FUNCTION_BLOCK FINAL FB_StepEngine EXTENDS FB_EventLogger  
VAR_INPUT
	Size					: UINT;
	Flags					: DWORD;
END_VAR             		
VAR_IN_OUT 
	Control					: ST_System;
	StepDesc				: ARRAY[*] OF STRING;
	MatrixA					: ARRAY[*] OF DINT;
	MatrixB					: ARRAY[*] OF DINT;
	MatrixC					: ARRAY[*] OF DINT;
	MatrixD					: ARRAY[*] OF DINT;
	TimerSP					: ARRAY[*] OF REAL;         		
END_VAR  
VAR_OUTPUT          		
	Outputs					: ARRAY[0..3] OF DINT; 
END_VAR             		
VAR      
	_StepReq				: INT;
	_DeviceAlarm			: BOOL;      		
	_SeqInterface			: ST_SequenceInterface;         		
	_StepTimeDn				: BOOL;
	_StepTimeRun			: BOOL;
	_StepChanged			: BOOL;
	_Disabled				: BOOL;
	_StepNum				: INT;
	_StepNumChan			: INT;
	_StepNumPrev			: INT;
	_StepTime_ET			: REAL;
	_StepTime_ETDT			: TIME;
	_StepTimeLeft			: REAL;
	_StepTimeLeftDT			: TIME;
	_StepTimePrev_ET		: REAL;
	_Message				: STRING;
	_Alarm					: BOOL;	
	_AlarmNum				: DINT;					
	_Fault					: BOOL;									
	_CurrentStep			: ARRAY[0..255] OF BOOL;
	_HistoryIndex			: INT;
END_VAR             		
VAR PERSISTENT      	
	_Name					: STRING[15];				
	_Description			: STRING[40];	
	_Disable				: BOOL;   			
	_AlarmMute				: BOOL;						
	_StepTime_PT			: REAL;
	_LastActiveStep			: INT;
	_History				: ARRAY[0..99] OF ST_SequenceHistory;	
	_Variables				: ARRAY [0..9] OF ST_Variable;									
END_VAR

M_AlarmMonitor();
F_CheckIndexBounds(0,UINT_TO_INT(Size),_StepNum);
F_CheckIndexBounds_REAL(0,65534,_StepTime_ET);
F_CheckIndexBounds_REAL(0,65534,_StepTime_PT);
F_CheckIndexBounds_REAL(0,65534,_StepTimeLeft);

IF  _Disable THEN
	_StepNum := 0;
	_Disabled := TRUE;
	_Message := 'Sequence Disabled';
ELSE
	_StepNum := _StepReq;
	_Disabled := FALSE;
	_Message:= StepDesc[_StepNum];
END_IF

IF Control.PackMLState.Complete THEN
	_LastActiveStep := 0;
END_IF

Outputs[0] := MatrixA[_StepNum];
Outputs[1] := MatrixB[_StepNum];
Outputs[2] := MatrixC[_StepNum];
Outputs[3] := MatrixD[_StepNum];

MEMSET(destAddr:= ADR(_CurrentStep), fillByte:= 0, n:= SIZEOF(_CurrentStep));
_CurrentStep[_StepNum] := TRUE;

IF _StepChanged THEN
	_StepTime_PT := TimerSP[_StepNum];
END_IF

_StepTime_ET := _StepTime_ET + Control.SystemTime.ScanTime;
_StepTime_ETDT := REAL_TO_TIME(_StepTime_ET);

IF _StepNum <> _StepNumChan THEN
	_StepTimePrev_ET := _StepTime_ET;
	_StepTime_ET := 0;
	_StepNumPrev := _StepNumChan;
	IF MatrixA[_StepNumChan].31 = TRUE THEN _LastActiveStep := _StepNumChan; END_IF
	IF MatrixA[_StepNumChan].30 = TRUE THEN _LastActiveStep := 0; END_IF	
	_StepNumChan := _StepNum;
	_StepChanged := TRUE;
	_StepTimeDn := FALSE;	
ELSE
	IF _StepTime_ET <= _StepTime_PT THEN
		_StepTimeLeft := _StepTime_PT - _StepTime_ET;
		_StepTimeLeftDT := REAL_TO_TIME(_StepTimeLeft);
	ELSE
		_StepTimeDn := TRUE;
	END_IF
	_StepChanged := FALSE;	
END_IF

IF _StepTime_PT = 0 THEN
	_StepTimeLeft := 0;
	_StepTimeLeftDT := REAL_TO_TIME(_StepTimeLeft);
END_IF

_History[0].StepNum:= _StepNum;
_History[0].StepTime:= _StepTime_ET;
_History[0].Message:= _Message;
	
IF _StepNumPrev <> _History[1].StepNum THEN 
	FOR _historyIndex:= 99 TO 2 BY -1 DO
		_History[F_CheckIndexBounds(0,99,_historyIndex)]:= _History[F_CheckIndexBounds(0,99,_historyIndex)-1];
	END_FOR
	_History[1].StepNum:= _StepNumPrev;
	_History[1].StepTime:= _StepTimePrev_ET;
	_History[1].Message:= StepDesc[_StepNumPrev];
END_IF

{attribute 'monitoring' := 'variable'}
PROPERTY PUBLIC Alarm : Bool
GET
Alarm := _Alarm;
END_GET
END_PROPERTY

{attribute 'monitoring' := 'variable'}
PROPERTY PUBLIC AlarmMute : BOOL
SET
AlarmMute := _AlarmMute;
END_SET
END_PROPERTY

{attribute 'monitoring' := 'variable'}
PROPERTY PUBLIC CurrentStep : REFERENCE TO ARRAY[0..255] OF BOOL
GET
CurrentStep REF= _CurrentStep;
END_GET
END_PROPERTY

{attribute 'monitoring' := 'variable'}
PROPERTY PUBLIC Description : String[40]
GET
Description := _Description;
END_GET
SET
_Description := Description;
END_SET
END_PROPERTY

{attribute 'monitoring' := 'variable'}
PROPERTY PUBLIC DeviceAlarm : BOOL
GET
DeviceAlarm :=_DeviceAlarm;
END_GET
SET
_DeviceAlarm := DeviceAlarm;
END_SET
END_PROPERTY

{attribute 'monitoring' := 'variable'}
PROPERTY PUBLIC Disable : BOOL
SET
_Disable := Disable;
END_SET
END_PROPERTY

{attribute 'monitoring' := 'variable'}
PROPERTY PUBLIC Disabled : BOOL
GET // PUBLIC
Disabled := _Disabled;
END_GET
SET
_Disabled := Disabled;
END_SET
END_PROPERTY

{attribute 'monitoring' := 'variable'}
PROPERTY PUBLIC Fault : Bool
SET
_Fault := Fault;
END_SET
END_PROPERTY

PROPERTY PUBLIC History :REFERENCE to ARRAY[0..99] OF ST_SequenceHistory
GET
History REF=_History;
END_GET
END_PROPERTY

{attribute 'monitoring' := 'variable'}
PROPERTY PUBLIC LastActiveStep : int
GET // PUBLIC
LastActiveStep := _LastActiveStep;
END_GET
SET
_LastActiveStep := LastActiveStep;
END_SET
END_PROPERTY

METHOD PROTECTED M_AlarmMonitor
VAR_INPUT
END_VAR
VAR_INST
END_VAR
VAR_INST // added by the converter: edge detectors and wires of the graphical bodies
    _w1, _w2 : BOOL;
END_VAR
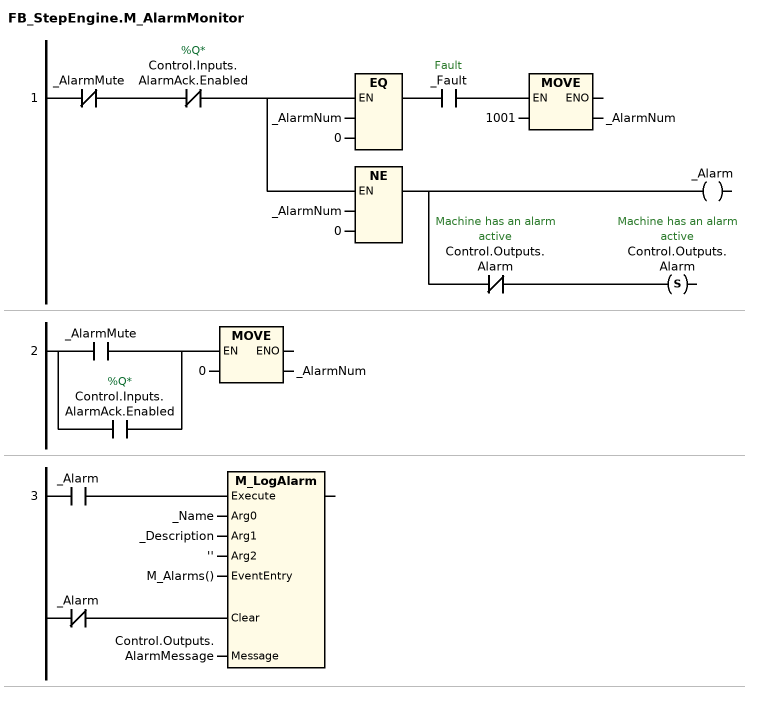
// NETWORK 1
//   Control.Inputs.AlarmAck.Enabled: AT %Q*
//   _Fault: Fault
//   Control.Outputs.Alarm: Machine has an alarm active
_w1 := NOT _AlarmMute AND NOT Control.Inputs.AlarmAck.Enabled;
IF (_w1 AND _AlarmNum = 0) AND _Fault THEN _AlarmNum := 1001; END_IF
_w2 := _w1 AND _AlarmNum <> 0;
_Alarm := _w2;
Control.Outputs.Alarm S= _w2 AND NOT Control.Outputs.Alarm;

// NETWORK 2
//   Control.Inputs.AlarmAck.Enabled: AT %Q*
IF _AlarmMute OR Control.Inputs.AlarmAck.Enabled THEN _AlarmNum := 0; END_IF

// NETWORK 3
M_LogAlarm(Execute := _Alarm, Arg0 := _Name, Arg1 := _Description, Arg2 := '', EventEntry := M_Alarms(), Clear := NOT _Alarm, Message := Control.Outputs.AlarmMessage);
END_METHOD

METHOD PRIVATE M_Alarms : TcEventEntry
VAR_INPUT
END_VAR
CASE _AlarmNum OF
	1001: M_Alarms:= TC_Events.TcSequence.A_1001;//Failed to Reach Requested State		
ELSE
	M_Alarms:= TC_Events.TcSequence.A_Undefined;
END_CASE
END_METHOD

{attribute 'monitoring' := 'variable'}
PROPERTY PUBLIC Name : String[15]
GET
Name := _Name;
END_GET
SET
_Name := Name;
END_SET
END_PROPERTY

{attribute 'monitoring' := 'variable'}
PROPERTY PUBLIC SeqInterface : REFERENCE TO ST_SequenceInterface
GET
SeqInterface REF= _SeqInterface;
END_GET
SET
_SeqInterface := SeqInterface;
END_SET
END_PROPERTY

{attribute 'monitoring' := 'variable'}
PROPERTY PUBLIC StepNum : INT
GET // PUBLIC
StepNum := _StepNum;
END_GET
SET // PUBLIC
_StepNum := StepNum;
END_SET
END_PROPERTY

{attribute 'monitoring' := 'variable'}
PROPERTY PUBLIC StepReq : INT
GET
StepReq := _StepReq;
END_GET
SET
_StepReq := StepReq;
END_SET
END_PROPERTY

{attribute 'monitoring' := 'variable'}
PROPERTY PUBLIC StepTime_ET : REAL
GET // PUBLIC
StepTime_ET := _StepTime_ET;
END_GET
END_PROPERTY

{attribute 'monitoring' := 'variable'}
PROPERTY PUBLIC StepTimeDn : BOOL
GET
StepTimeDn := _StepTimeDn;
END_GET
END_PROPERTY

PROPERTY PUBLIC Variables : REFERENCE TO ARRAY[0..9] OF ST_Variable
GET
Variables REF= _Variables;
END_GET
END_PROPERTY

END_FUNCTION_BLOCK

(* stored: Version 1.1.0.1, ProductVersion 3.1.4024.3
   POU FB_StepEngine: Id {4fdbb4a1-3842-443f-89c2-dd769aeef5ad}, SpecialFunc None
   Property Alarm: Id {837ab50d-3215-4ed0-a93e-6651d97b3d28}
   Get Get: Id {1c9c6dfd-b4ce-4428-9ce9-6c2f1ac6a132}
   Property AlarmMute: Id {160223e5-9e2d-4eaa-81d1-9adae92b6c4c}
   Set Set: Id {68a96057-a0af-4e79-84c1-e6ba000028f6}
   Property CurrentStep: Id {2037412a-16f8-47af-af3e-793245d8f6a9}
   Get Get: Id {39dda43d-52af-4f86-8bbb-681aa9fe8c87}
   Property Description: Id {0f1f32f0-a82c-461c-a727-547d7f793953}
   Get Get: Id {90b27f05-48cd-4083-b14e-adf2035350be}
   Set Set: Id {37617139-61e1-44f0-b9b5-a6a1d7b28a26}
   Property DeviceAlarm: Id {3bc8205d-08de-448b-8620-de355da933cc}
   Get Get: Id {7738ded8-563d-403e-a885-d4480570b89e}
   Set Set: Id {60d9ec6b-e6ec-43fd-9fe0-328014683f9d}
   Property Disable: Id {aaf760da-0cc1-4549-8735-8ee60af60cd8}
   Set Set: Id {c89da68e-aec3-4029-aca2-5ee35067ee60}
   Property Disabled: Id {5d573e8b-ce38-485d-9f8a-3f2d68a5acd2}
   Get Get: Id {a218fcc3-ce98-4739-9a41-dced224b0dc7}
   Set Set: Id {53537a12-e145-4039-aba4-0db12406a856}
   Property Fault: Id {6ad063fc-0083-4977-8f2c-d2c052a23fa9}
   Set Set: Id {98a1f858-3f84-4b6f-b0e2-1522fc22fb4b}
   Property History: Id {47d47c1c-f340-4bed-85ea-8cc19a900daf}
   Get Get: Id {80016576-c89b-4cee-a2bb-2d6f914e144d}
   Property LastActiveStep: Id {b4a1b963-433c-4a05-ac2d-c168021af49c}
   Get Get: Id {c69b5b85-481f-48a0-9b99-b5c13dd85c40}
   Set Set: Id {b94674cd-6e96-4dea-8b76-c024cde67b82}
   Method M_AlarmMonitor: Id {e08c103d-6dec-40ba-9878-824a65d1445f}
   Method M_Alarms: Id {9108062e-d719-441f-a857-223fc164f81e}
   Property Name: Id {da780c25-1ea0-4d2a-9645-691f350a0148}
   Get Get: Id {1ee78ae4-6d76-4f8b-89d0-55735eee87d9}
   Set Set: Id {a9538816-0b8e-46ec-8164-f2194c4c23ed}
   Property SeqInterface: Id {c5867ce7-dc85-4a63-8151-f52b897b5d59}
   Get Get: Id {c6129851-ed72-4d44-8bd1-eee06b4a27de}
   Set Set: Id {a8d65edd-cd08-4e9d-8239-c7534116fce9}
   Property StepNum: Id {130bd683-47ea-4e90-b3ab-f858e4d60918}
   Get Get: Id {75f3e48c-3d37-423b-a9b1-ebaf6fcfdb42}
   Set Set: Id {3a11944c-db0a-4cdc-8b7d-038bde4b44c7}
   Property StepReq: Id {fae1f7a4-307c-418d-8568-ae40f3e9ac87}
   Get Get: Id {9c14fa1a-19f9-4db6-9412-c6dfa1031b2c}
   Set Set: Id {980128ab-b28e-419c-83d8-b7955cf5cf62}
   Property StepTime_ET: Id {995ecc46-0c06-4057-abe1-bf793c0b67cd}
   Get Get: Id {03f2c4b2-2a2f-47c0-9595-9f454de1030e}
   Property StepTimeDn: Id {6e4618c3-946e-4e6f-9a8d-eda670e7295b}
   Get Get: Id {dafd0d52-a2e6-4f7b-a05b-69f3654182d3}
   Property Variables: Id {12c62f2c-42f0-4fb4-bc9f-c6c10455f5ea}
   Get Get: Id {5c78cd74-ff17-44ff-9b2d-747709c179d7} *)
